Staubli VAL3: TrajBypass.pgx

public program TrajBypass(bool& x_bByPass (dimensions=1), num x_nIndex (dimensions=1))
begin

  //通过外围信号来对路径是否生产进行判断

  aioSet(aAio["O2_aNull"],x_nIndex)
  logMsg("等待信号"+toString("",x_nIndex)+"路径是否过滤")

  //信号自定义
  //仅仅作为测试使用
  //  wait(aioGet(aAio["In4_a7CurPosH"])==x_nIndex)
  //  x_bByPass=(dDio["In1_bNull1"]==true)

end
